FUNCTION Greater_Smaller
VAR_INPUT
	nNumber1 : INT;
	nNumber2 : INT;
END_VAR
VAR_OUTPUT
	nGreater : INT;
	nSmaller : INT;
END_VAR

IF nNumber1 > nNumber2 THEN
	nGreater := nNumber1;
	nSmaller := nNumber2;
ELSE
	nGreater := nNumber2;
	nSmaller := nNumber1;
END_IF

END_FUNCTION

(* stored: Version 1.1.0.1, ProductVersion 3.1.4024.11
   POU Greater_Smaller: Id {da9d3f4e-d593-44a3-b23d-2eca1b63a823}, SpecialFunc None *)
